{attribute 'OPC.UA.DA' := '0'}
TYPE LsCalibrateConfig :
STRUCT
	HSPowermeter : HSPowermeter;
	HTPowermeter : HTPowermeter;
END_STRUCT
END_TYPE

(* stored: Version 1.1.0.1, ProductVersion 3.1.4024.4
   DUT LsCalibrateConfig: Id {c813de1b-4345-4547-8cee-14addd1cc236} *)
